# EPICS substitutions: apps/jscalerApp/Db/jscalers_ftc_quadrant.substitutions
file "db/jscalers_ftc_quadrant.template" {
pattern
{Q X01 X02 X03 X04 X05 X06 X07 X08 X09 X10 X11 Y12 Y13 Y14 Y15 Y16 Y17 Y18 Y19 Y20 Y21 Y22}
{1  01  02  03  04  05  06  07  08  09  10  11  12  13  14  15  16  17  18  19  20  21  22}
{2  22  21  20  19  18  17  16  15  14  13  12  12  13  14  15  16  17  18  19  20  21  22}
{3  22  21  20  19  18  17  16  15  14  13  12  11  10  09  08  07  06  05  04  03  02  01}
{4  01  02  03  04  05  06  07  08  09  10  11  11  10  09  08  07  06  05  04  03  02  01}
}
